FUNCTION_BLOCK TcoDigitalInspectorTests EXTENDS TcoCore._internals_TcoContext
VAR
    _sut            : TcoInspectors.TcoDigitalInspector(THIS^);
    _inspectedValue : BOOL;
    _result         : TcoInspectors.eInspectorResult;
    _isOverIspected : BOOL;
    _overallResult  : TcoInspectors.TcoComprehensiveResult;
END_VAR

METHOD PROTECTED Main
CASE _testId OF
    0:
        _result         := 0;
        _isOverIspected := FALSE;
    eDigitalInspectorTests.Inspect:
        THIS^.ProbeDoneWhen(_sut.Inspect(_inspectedValue).UpdateComprehensiveResult(_overallResult).Done);	
    eDigitalInspectorTests.GetResult:
        _result         := _sut.Inspect(_inspectedValue).Result;
        _isOverIspected := _sut.Inspect(_inspectedValue).OverInspected;						
END_CASE
END_METHOD

END_FUNCTION_BLOCK

(* stored: Version 1.1.0.1, ProductVersion 3.1.4024.9
   POU TcoDigitalInspectorTests: Id {8e88c5fb-6b37-0ee0-1dee-44bcdb0de8e4}, SpecialFunc None
   Method Main: Id {2386eb08-ae25-07fa-0ae2-18bdce87e272} *)
